Staubli VAL3: page.pgx

public program page(string& menuname[], num index)
// set all the page in english
begin
  //
  //  PAGE
  //
  //
  // PALLET PAGE
  if index>=10 and index<=19
    title("< Page Pallet >")
  endIf
  // PALLET VIEW PAGE
  if index>=100 and index<=109
    title("< Page View Pallet >")
  endIf
  switch index
    //
    // PALLET
    //
    // Integrator programmer
    case 10,11
      menuname="View Program,Edit Pallet,,,Wizard,Reset,Back,Next"
    break
    // On Cycle
    case 13,14
      menuname="View Program,Edit Pallet,,,,Reset,Back,Next"
    break
    // VIEW PALLET
    case 100,101,102,103,104,105
      menuname="Reset ALL,,,,,Reset,Back,Next"
    break
  endSwitch
end
